FUNCTION_BLOCK RefeedingConveyor EXTENDS Conveyor
VAR_INPUT
END_VAR
VAR_OUTPUT
END_VAR
VAR
	//Sensors
	m_PresencesensorStart : PresenceSensor;
	m_PresencesensorEnd : PresenceSensor;
	
	//Pusher
	m_Switch : Switch;
END_VAR

METHOD METH_Switch_Extend : BOOL
VAR_INPUT
END_VAR
m_Switch.METH_Extend();
END_METHOD

METHOD METH_Switch_Retract : BOOL
VAR_INPUT
END_VAR
m_Switch.METH_Retract();
END_METHOD

PROPERTY WPAtEnd : BOOL
GET
WPAtEnd := m_PresencesensorEnd.Value;
END_GET
END_PROPERTY

PROPERTY WPAtStart : BOOL
GET
WPAtStart := m_PresencesensorStart.Value;
END_GET
END_PROPERTY

END_FUNCTION_BLOCK

(* stored: Version 1.1.0.1
   POU RefeedingConveyor: Id {f41b28dd-09bf-4ed8-8981-8099f0126724}, SpecialFunc None
   Folder Methods: Id {20dc8d37-440a-4538-af0b-c58f24985255}
   Folder Properties: Id {08741579-5da2-431c-99b0-57c0dcb55c09}
   Method METH_Switch_Extend: Id {49aff4b8-42d1-46cd-8d19-e98540bd4035}
   Method METH_Switch_Retract: Id {12b3bddf-7376-43d1-b82f-66513aaf06ee}
   Property WPAtEnd: Id {405b0475-9370-4864-a42e-f714bdbbebdf}
   Get Get: Id {bd1eac21-9f42-4327-8a22-809463bbf012}
   Property WPAtStart: Id {a0f1eb6a-5ede-4b93-96d6-b1b7a587b255}
   Get Get: Id {882960c9-946e-430f-bf9d-016dbd15efd7} *)
